PROGRAM StandardCPM
VAR
	ProdStd : REAL;
	BriteCode_Standards : StandardCPMSet;
END_VAR

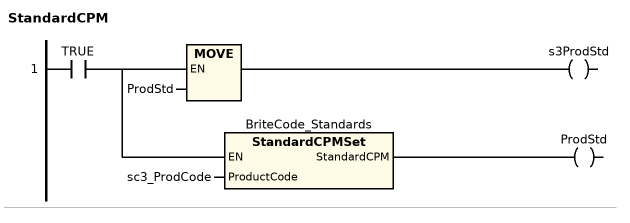
// NETWORK 1
s3ProdStd := ProdStd;
BriteCode_Standards(ProductCode := sc3_ProdCode); // StandardCPMSet
ProdStd := BriteCode_Standards.StandardCPM;

END_PROGRAM

(* stored: Version 1.1.0.1, ProductVersion 3.1.4024.15
   POU StandardCPM: Id {ee5f6ead-8b1a-4243-9215-d141a9286faa}, SpecialFunc None *)
